(* PLC project Modbus_Test_Project.project, CODESYS CODESYS V3.5 SP20 Patch 5 *)
(* stored: creationDateTime 2025-06-30T17:58:16.8976783, modificationDateTime 2025-06-25T17:03:43.3271085 *)

PROGRAM Main
  VAR
    modbusSlave : FB_ModbusSlave;
  END_VAR

                    modbusSlave();
                  
END_PROGRAM

FUNCTION_BLOCK FB_ModbusSlave
  VAR
    aDiscreteInputsMemory : ARRAY[0..9] OF BOOL;
    aCoilsMemory1 : ARRAY[0..4] OF BOOL;
    aCoilsMemory2 : ARRAY[0..4] OF BOOL;
    aInputRegistersMemory1 : ARRAY[0..6] OF UINT;
    aInputRegistersMemory2 : ARRAY[0..2] OF UINT;
    aHoldingRegistersMemory : ARRAY[0..6] OF UINT;
  END_VAR
  VAR CONSTANT
    fcsSupported : ModbusFB.SupportedFcs := (ReadCoils := TRUE, ReadDiscreteInputs := TRUE, ReadHoldingRegisters := TRUE, ReadInputRegisters := TRUE, WriteSingleCoil := TRUE, WriteSingleRegister := TRUE);  (* custom defined fcsSupported *)
    aDiscreteInputsSections : ARRAY[0..0] OF ModbusFB.TableSection := [(uiStart := 0, uiNumDataItems := 10, pStartAddr := ADR(aDiscreteInputsMemory[0]), uiDataItemSize := 8)];  (* Simple multi-section "data model". This "data model" is completely memory mapped (all "data items" mapped to memory). It contains non-consecutive "data items" and non-consecutive data item memory to demonstrate how to setup such a configuration. "plain vanilla" setup can be done also, see "discrete inputs". "discrete inputs" - "plain vanilla": consecutive "data items" (0..n-1) and consecutive data item memory (one block of memory for all "data items"). *)
    aCoilsSections : ARRAY[0..1] OF ModbusFB.TableSection := [(uiStart := 0, uiNumDataItems := 5, pStartAddr := ADR(aCoilsMemory1[0]), uiDataItemSize := 8), (uiStart := 5, uiNumDataItems := 5, pStartAddr := ADR(aCoilsMemory2[0]), uiDataItemSize := 8)];  (* "coils" - consecutive "data items" and non-consecutive data item memory *)
    aInputRegistersSections : ARRAY[0..2] OF ModbusFB.TableSection := [(uiStart := 0, uiNumDataItems := 3, pStartAddr := ADR(aInputRegistersMemory1[0]), uiDataItemSize := 16), (uiStart := 5, uiNumDataItems := 4, pStartAddr := ADR(aInputRegistersMemory1[3]), uiDataItemSize := 16), (uiStart := 10, uiNumDataItems := 3, pStartAddr := ADR(aInputRegistersMemory2[0]), uiDataItemSize := 16)];  (* "input registers" - non-consecutive "data items" and non-consecutive data item memory *)
    aHoldingRegistersSections : ARRAY[0..1] OF ModbusFB.TableSection := [(uiStart := 0, uiNumDataItems := 6, pStartAddr := ADR(aHoldingRegistersMemory[0]), uiDataItemSize := 16), (uiStart := 7, uiNumDataItems := 3, pStartAddr := ADR(aInputRegistersMemory2[0]), uiDataItemSize := 16)];  (* "holding registers" - consecutive "data items" and consecutive data item memory "holding registers" 7..9 overlap with "input registers" 10..12 *)
    tableDefs : ModbusFB.TableDefinitions := (tableDiscreteInputs := (uiNumSections := 1, pSections := ADR(aDiscreteInputsSections[0])), tableCoils := (uiNumSections := 2, pSections := ADR(aCoilsSections[0])), tableInputRegisters := (uiNumSections := 3, pSections := ADR(aInputRegistersSections[0])), tableHoldingRegisters := (uiNumSections := 2, pSections := ADR(aHoldingRegistersSections[0])));  (* the "data model" tables *)
  END_VAR
  VAR
    serverTCP : ModbusFB.ServerTCP;  (* our MODBUS TCP server (slave) *)
    serverSerial : ModbusFB.ServerSerial;  (* our MODBUS RTU server (slave) *)
    initDone : BOOL := FALSE;
  END_VAR

                    IF NOT initDone THEN
	initDone := TRUE;
	// configure tcpServer 
	serverTCP(fcsSupported:=fcsSupported, dataModel:=tableDefs, wsInterfaceName:="", uiPort:=1100);
	// configure serialServer 
END_IF

// call the server FB's
serverTCP(xEnable:=TRUE);
serverSerial(xEnable:=TRUE);


 

                  
END_FUNCTION_BLOCK

CONFIGURATION CODESYS_Control_Win_V3
  RESOURCE Application ON PLC
    TASK Task(INTERVAL := T#20ms, PRIORITY := 1);
    PROGRAM Main WITH Task : Main;
  END_RESOURCE
END_CONFIGURATION
